// TIA Portal V16 export
// export: Created 2021-07-12T14:47:21.2092262Z, ExportSetting WithDefaults, DisplayName Totally Integrated Automation Portal, DisplayVersion V16, DisplayName TIA Portal Version Control Interface, DisplayVersion V16, DisplayName TIA Portal Openness, DisplayVersion V16, DisplayName STEP 7 Professional, DisplayVersion V16, DisplayName STEP 7 Safety, DisplayVersion V16, DisplayName WinCC Professional, DisplayVersion V16
TYPE "SimaHydTO_typeHMIConnectionParameterSettings"
TITLE = SimaHydTO_typeHMIConnectionParameterSettings
// HMI interface: Parameter settings
// stored: IsFailsafeCompliant false
   STRUCT
      AxisData { S7_SetPoint := 'True'} : "SimaHydTO_typeHMIConnectionParameterSettingsAxisData";
      Commands { S7_SetPoint := 'True'} : "SimaHydTO_typeHMIConnectionParameterSettingsCommands";   // Data: HMI -> PLC
      Status { S7_SetPoint := 'True'} : "SimaHydTO_typeHMIConnectionParameterSettingsStatus";   // Data: PLC -> HMI
   END_STRUCT;
END_TYPE
